(* IEC 61131-3 sources: ArfBotOS/Codesys-4/ArfBotOS.fbsdev/Application.iecapp^/FUN/controller/FB_Controller.fb.st^/public, 7 files *)

(* ---- M_SetBrightness.meth.st ---- *)
METHOD PUBLIC M_SetBrightness : BOOL
VAR_INPUT
	Brightness: E_ControllerBrightness;
END_VAR

M_SetBrightness := TRUE;
_Brightness := Brightness;
_SetBrightness := TRUE;
END_METHOD

(* ---- M_SetColor.meth.st ---- *)
METHOD PUBLIC M_SetColor : BOOL
VAR_INPUT
	Red: INT:=0;
	Green: INT:=255;
	Blue: INT:=0;
END_VAR

IF Red>=0 AND_THEN Red<=255
	AND_THEN Green>=0 AND_THEN Green<=255
	AND_THEN Blue>=0 AND_THEN Blue<=255THEN
		M_SetColor := TRUE;
		_SetColor:=TRUE;
		_Red:=Red;
		_Green:=Green;
		_Blue:=Blue;
ELSE
	M_SetColor := FALSE;
END_IF
END_METHOD

(* ---- M_SetMicrophoneState.meth.st ---- *)
METHOD PUBLIC M_SetMicrophoneState : BOOL
VAR_INPUT
	State: BOOL;
END_VAR

M_SetMicrophoneState := TRUE;
_MicrophoneState := State;
_SetMicrophoneState := TRUE;
END_METHOD

(* ---- M_SetMotorIntensity.meth.st ---- *)
METHOD PUBLIC M_SetMotorIntensity : BOOL
VAR_INPUT
	Motor: E_ControllerMotor;
	Intensity: USINT; // 0-255
	Duration: REAL; // s
END_VAR

IF Intensity >=0 AND_THEN Intensity <= 255 AND_THEN Duration <= 5000 THEN
	M_SetMotorIntensity := TRUE;
	_SetMotorIntensity := TRUE;
	_Motor := Motor;
	_MotorIntensity := Intensity;
	_MotorIntensityDuration := Duration;
ELSE
	M_SetMotorIntensity := FALSE;
END_IF
END_METHOD

(* ---- M_SetPlayerID.meth.st ---- *)
METHOD PUBLIC M_SetPlayerID : BOOL
VAR_INPUT
	PlayerID: E_ControllerPlayerID;
END_VAR

M_SetPlayerID := TRUE;
_PlayerID := PlayerID;
_SetPlayerID := TRUE;
END_METHOD

(* ---- M_SetTriggerForce.meth.st ---- *)
METHOD PUBLIC M_SetTriggerForce : BOOL
VAR_INPUT
	Trigger: E_ControllerTrigger;
	Parameter: E_ControllerTriggerForceParameter;
	Intensity: USINT; // 0-255
END_VAR

IF Intensity >= 0 AND Intensity <= 255 THEN
	M_SetTriggerForce := TRUE;
	_SetTriggerForce:=TRUE;
	_TriggerForceTrigger := Trigger;
	_TriggerForceParameter := Parameter;
	_TriggerForceIntensity := Intensity;
ELSE
	M_SetTriggerForce := FALSE;
END_IF
END_METHOD

(* ---- M_SetTriggerMode.meth.st ---- *)
METHOD PUBLIC M_SetTriggerMode : BOOL
VAR_INPUT
	Trigger: E_ControllerTrigger;
	Mode: E_ControllerTriggerMode;
END_VAR

M_SetTriggerMode := TRUE;
_SetTriggerMode := TRUE;
_TriggerModeTrigger := Trigger;
_TriggerModeMode := Mode;
END_METHOD
